Fanuc KAREL source: ka00077.KL

-- PROVISIONAL review KL for V940-1; original PC SHA256 0e2a7994a3b022c1463cdff19aee66dfdba6340b6d8e78dbcd53e1354faea04d
-- Incomplete behavior may be omitted. Consult companion uncertainty JSON. Do not deploy.
PROGRAM KA00077
%NOLOCKGROUP
-- UNRESOLVED_DECL SRC type=000106
-- UNRESOLVED_DECL DST type=000101
BEGIN
  -- V9_ZERO_TABLE_METADATA_HINT layout=0001; no indexed target words; source/name/runtime held
  -- UNRESOLVED_PC offsets 5-20; opcodes 2E,22,32,35
  -- UNRESOLVED_PC offsets 25-45; opcodes 49,7E,4A
  -- UNRESOLVED_PC offsets 50-54; opcodes 7F
END KA00077
